(* IEC 61131-3 sources: generating_plc_code_with_llms/PLC_Code, 21 files *)

(* ---- 10.st ---- *)
FUNCTION SIGMOID : REAL
  VAR_INPUT
    X : REAL;
  END_VAR

  IF X > 20.0 THEN
  	SIGMOID := 1.0;
  ELSIF x < -85.0 THEN
  	SIGMOID := 0.0;
  ELSE
  	SIGMOID := 1.0 / (1.0 + EXP(-X));
  END_IF;
  (* from OSCAT library; www.oscat.de  *)
END_FUNCTION

(* ---- 11.st ---- *)
FUNCTION SGN : INT
  VAR_INPUT
    x : REAL;
  END_VAR

  IF X > 0.0 THEN
  	sgn := 1;
  ELSIF X < 0.0 THEN
  	sgn := -1;
  ELSE
  	sgn := 0;
  END_IF;
  (* from OSCAT library; www.oscat.de  *)
END_FUNCTION

(* ---- 12.st ---- *)
FUNCTION SINH : REAL
  VAR
    X : REAL;
  END_VAR

  IF ABS(x) < 2.0E-3 THEN
  	SINH := X;
  ELSE
  	SINH := (EXP(x) - EXP(-x)) * 0.5;
  END_IF;
  (* from OSCAT library; www.oscat.de  *)
END_FUNCTION

(* ---- 14.st ---- *)
FUNCTION FC1001 :BOOL
VAR_INPUT
	MEW: REAL;
	SP: REAL;
	HYS: REAL;
END_VAR
VAR_IN_OUT
 	OUT:BOOL;
END_VAR
VAR
 	P_HYS: REAL;
END_VAR

P_HYS:=MEW*HYS/100;
IF MEW<(SP-P_HYS/2) THEN
	OUT:=TRUE;
ELSIF
	MEW>(SP+P_HYS/2) THEN
	OUT:=FALSE;
ELSE
	OUT:=OUT;
END_IF

(* ---- 15.st ---- *)
FUNCTION FC1002 :BOOL
VAR_INPUT
	E_A, SENSOR: BOOL;
	ZEITW: TIME;
END_VAR
VAR_IN_OUT
	ZEIT:TON;
	P_HU, P_AL: BOOL;
END_VAR

IF NOT E_A THEN
	FC1002:=FALSE;
	P_HU:=FALSE;
	P_AL:=FALSE;
ELSE
	FC1002:=TRUE;
	IF P_AL THEN
		P_HU:=FALSE;
	ELSIF SENSOR THEN
		P_HU:=FALSE;
	ELSE
		P_HU:=TRUE;
	END_IF
END_IF
ZEIT(IN:=P_HU OR P_AL, PT:=ZEITW);
P_AL:=Zeit.Q;

(* ---- 18.st ---- *)
FUNCTION FC1003 : VOID
VAR_INPUT
    IN_R:REAL;
    IN_MAX, IN_MIN:REAL;
    OUT_MAX, OUT_MIN:REAL;
END_VAR
VAR_OUTPUT
    OUT_R:REAL;
    FEH:BOOL;
END_VAR
VAR_TEMP
    DIFF1, DIFF2:REAL;
END_VAR

DIFF1:= IN_MAX-IN_MIN;
DIFF2:= OUT_MAX-OUT_MIN;
FEH := (DIFF1=0) OR (DIFF2=0);
IF NOT FEH THEN
    OUT_R:= (OUT_MAX-OUT_MIN) / DIFF1 * (IN_R-IN_MIN) + OUT_MIN;
ELSE
    OUT_R:=0.0;
END_IF;
END_FUNCTION

(* ---- 2.st ---- *)
FUNCTION BINOM : INT
  VAR_INPUT
    N : INT;
    K : INT;
    i : INT;
  END_VAR

  IF 2 * K > n THEN
  	k := n - k;
  END_IF;
  IF k > n THEN
  	RETURN;
  ELSIF k = 0 OR k = n THEN
  	BINOM := 1;
  ELSIF k = 1 THEN
  	BINOM := n;
  ELSE
  	BINOM := n;
  	n := n + 1;
  	FOR i := 2 TO k DO
  		BINOM := BINOM * (n - i) / i;
  	END_FOR;
  END_IF;

END_FUNCTION

(* ---- 3.st ---- *)
FUNCTION FIB : DINT
  VAR_INPUT
    X : INT;
  END_VAR
  VAR
    t1 : DINT;
    t2 : DINT;
    x_tmp : INT;
  END_VAR

  t1 := DINT#0;
  t2 := DINT#0;
  X_tmp := X;
  IF X_tmp < 0 OR X_tmp > 46 THEN
  	FIB := DINT#-1;
  ELSIF X_tmp < 2 THEN
  	FIB := INT_TO_DINT(X_tmp);
  	RETURN;
  ELSE
  	(* the fibonacci number is the sum of the two suceeding fibonaci numbers *)
  	(* we store the numbers alternatively in t1 and t2 depending on pt *)
  	t2 := DINT#1;
  	WHILE X_tmp > 3 DO
  		X_tmp := X_tmp - 2;
  		t1 := t1 + t2;
  		t2 := t1 + t2;
  	END_WHILE;
  	IF X_tmp > 2 THEN t1 := t1 + t2; END_IF;
  	fib := t1 + t2;
  END_IF;
END_FUNCTION

(* ---- 8.st ---- *)
FUNCTION LAMBERT_W : REAL
  VAR_INPUT
    X : REAL;
  END_VAR
  VAR
    w : REAL;
    i : INT;
    we : REAL;
    w1e : REAL;
    ewx : REAL;
    last : DWORD;
  END_VAR

  IF x < -0.367879441171442 THEN
  	LAMBERT_W := -1000.0;
  	RETURN;
  (* return 0 if x = 0 *)
  ELSIF x = 0.0 THEN
  	RETURN;
  (* first an estimate is calculated *)
  ELSIF x <= 500.0 THEN
  	w := LN(x + 1.0);
  	w := 0.665 * (1.0 + 0.0195 * w) * w + 0.04;
  ELSE
  	w := LN(x - 4.0) - (1.0 - 1.0/LN(x)) * LN(LN(x));
  END_IF;
  (* use estimate to calculate exact result *)
  FOR i := 0 TO 5 DO
  	ewx := EXP(w);
  	we := w * ewx - x;
  	w1e := (w+1.0) * ewx;
  	last := REAL_TO_DWORD(w) AND DWORD#16#FFFF_FFFC;
  	w := w - (we / (w1e - (w+2.0) * we / (2.0 * w + 2.0)));
  	IF (REAL_TO_DWORD(w) AND DWORD#16#FFFF_FFFC) = last THEN EXIT; END_IF;
  END_FOR;
  LAMBERT_W := w;
  (* from OSCAT library; www.oscat.de  *)
END_FUNCTION

(* ---- 19.st ---- *)
FUNCTION_BLOCK FB1005
VAR_INPUT
    START:BOOL;
    DICKE, V_MAX, V_MIN:REAL;
END_VAR
VAR_OUTPUT
    D_MAX, D_MIN:REAL;
    P1:BOOL;
END_VAR
VAR
    FO:BOOL;
END_VAR

IF NOT START THEN
    FO:=START;
    RETURN;
END_IF;
IF START=TRUE AND FO=FALSE THEN
    D_MAX:=DICKE;
    D_MIN:=DICKE;
    P1:=FALSE;
END_IF;
FO:=START;
IF DICKE < D_MIN THEN
    D_MIN:=DICKE;
END_IF;
IF DICKE > D_MAX THEN
    D_MAX:=DICKE;
END_IF;
IF D_MIN < V_MIN OR D_MAX > V_MAX THEN
    P1:=TRUE;
END_IF;
END_FUNCTION_BLOCK

(* ---- 20.st ---- *)
FUNCTION_BLOCK INTERLOCK
    VAR_INPUT
        I1 : BOOL;
        I2 : BOOL;
        TL : TIME;
    END_VAR
    VAR_OUTPUT
        Q1 : BOOL;
        Q2 : BOOL;
    END_VAR
    VAR
        T1 : TOF;
        T2 : TOF;
    END_VAR

    T1(IN := I1, PT := TL);
    T2(IN := I2, PT := TL);

    Q1 := I1 AND NOT t2.Q;
    Q2 := I2 AND NOT t1.Q;

END_FUNCTION_BLOCK

(* ---- 21.st ---- *)
FUNCTION_BLOCK BURNER
  VAR_INPUT
    IN : BOOL;
    STAGE2 : BOOL;
    OVER_TEMP : BOOL;
    OIL_TEMP : BOOL := TRUE;
    FLAME : BOOL;
    RST : BOOL;
    RST_TIMER : BOOL;
    PRE_HEAT_TIME : TIME := t#5s;
    PRE_VENT_TIME : TIME := t#15s;
    PRE_IGNITE_TIME : TIME := t#15s;
    POST_IGNITE_TIME : TIME := t#25s;
    STAGE2_DELAY : TIME := t#10s;
    SAFETY_TIME : TIME := t#5s;
    LOCKOUT_TIME : TIME := t#10s;
    MULTIPLE_IGNITION : BOOL := TRUE;
    KW1 : REAL;
    KW2 : REAL;
  END_VAR
  VAR_OUTPUT
    MOTOR : BOOL;
    COIL1 : BOOL;
    COIL2 : BOOL;
    PRE_HEAT : BOOL;
    IGNITE : BOOL;
    FAIL : BOOL;
    KWH : REAL;
    STATUS : BYTE;
  END_VAR
  VAR_IN_OUT
    RUNTIME1 : UDINT;
    RUNTIME2 : UDINT;
    CYCLES : UDINT;
  END_VAR
  VAR
    state : INT;
    last : TIME;
    tx : TIME;
    last_change : TIME;
    timer1 : ONTIME;
    timer2 : ONTIME;
    oil_temp_last : BOOL;
    cycles2 : UDINT;
  END_VAR

  tx:= UDINT_TO_TIME(T_PLC_MS(en:=true));

  (* check rst input and overtemp *)
  IF rst OR over_temp OR state = 0 THEN
  	IF status > BYTE#0 AND tx - last_change >= lockout_time AND rst THEN
  		status := BYTE#110;
  		fail := FALSE;
  		state := 1;
  	ELSE
  		(* normaler reset *)
  		motor := FALSE;
  		coil1 := FALSE;
  		coil2 := FALSE;
  		ignite := FALSE;
  		pre_heat := FALSE;
  		IF over_temp THEN
  			status := BYTE#9;
  			fail := TRUE;
  		END_IF;
  		last_change := tx;
  		last := tx;
  		state := 1;
  	END_IF;
  END_IF;

  (* check for timer rst and rst timer if true *)
  IF rst_timer THEN
  	runtime1 := UDINT#0;
  	runtime2 := UDINT#0;
  	cycles := UDINT#0;
  	cycles2 := UDINT#0;
  END_IF;

  (* quit here if an error is present *)
  IF (status > BYTE#0 AND status < BYTE#100) OR rst THEN RETURN; END_IF;

  (* start sequence *)
  CASE state OF

  1:	(* in signal starts oil pre heating *)
  	IF in AND flame THEN
  		state := 7;
  		pre_heat := FALSE;
  		status := BYTE#2;
  		last_change := tx;
  	ELSIF in THEN
  		pre_heat := TRUE;
  		state := 2;
  		last_change := tx;
  	END_IF;

  2:	(* after pre_heating time start motor *)
  	IF (tx- last_change >= pre_heat_time AND oil_temp) OR (oil_temp AND NOT oil_temp_last) THEN
  		motor := TRUE;
  		state := 3;
  		last_change := tx;
  	(* pre_heat_time ist abgelaufen und oil_temp ist nicht aktiv *)
  	ELSIF tx - last_change >= pre_heat_time AND NOT oil_temp THEN
  		state := 7;
  		pre_heat := FALSE;
  		status := BYTE#1;
  		last_change := tx;
  	(* flame monitor cannot be active at this time *)
  	ELSIF flame THEN
  		state := 7;
  		pre_heat := FALSE;
  		status := BYTE#2;
  		last_change := tx;
  	END_IF;

  3:	(* abwarten bis zündung eingeschaltet werden kann *)
  	IF tx - last_change >= pre_vent_time - pre_ignite_time THEN
  		ignite := TRUE;
  		state := 4;
  		last_change := tx;
  	(* flame monitor cannot be active at this time *)
  	ELSIF flame THEN
  		state := 7;
  		pre_heat := FALSE;
  		motor := FALSE;
  		status := BYTE#3;
  		last_change := tx;
  	END_IF;

  4:	(* warten bis oelzufuhr geoeffnet werden darf *)
  	IF tx - last_change >= pre_ignite_time THEN
  		coil1 := TRUE;
  		state := 5;
  		last_change := tx;
  	END_IF;

  5:	(* warten auf flammwaechter und falls noetig abschalten *)
  	IF tx - last_change >= safety_time OR flame THEN
  		IF NOT flame THEN
  			(* notabschaltung da flammwaechster nicht angesprochen hat *)
  			state := 7;
  			motor := FALSE;
  			coil1 := FALSE;
  			pre_heat := FALSE;
  			ignite := FALSE;
  			status := BYTE#4;
  			last_change := tx;
  		ELSE
  			state := 6;
  			last_change := tx;
  		END_IF;
  	END_IF;

  6:	(* brenner läuft, flammueberwachung und nach ablauf der nachigniteszeit ignite abschalten *)
  	IF NOT flame AND NOT multiple_ignition THEN
  		(* notabschaltung da flammwaechster keine flamme meldet *)
  		state := 7;
  		motor := FALSE;
  		coil1 := FALSE;
  		coil2 := FALSE;
  		pre_heat := FALSE;
  		ignite := FALSE;
  		status := BYTE#5;
  		last_change := tx;
  	ELSIF NOT flame AND multiple_ignition THEN
  		ignite := TRUE;
  		state := 5;
  		coil2 := FALSE;
  		last_change := tx;
  	ELSE
  		IF tx - last_change >= post_ignite_time THEN
  			(* post_ignite_time abgelaufen, ignite abschalten *)
  			ignite := FALSE;
  		END_IF;
  		IF tx - last_change >= stage2_delay AND stage2 THEN
  			coil2 := TRUE;
  		ELSE
  			coil2 := FALSE;
  		END_IF;
  	END_IF;
  END_CASE;

  (* abschaltung wenn kein eingangssignal *)
  IF NOT in THEN
  	state := 1;
  	motor := FALSE;
  	coil1 := FALSE;
  	coil2 := FALSE;
  	ignite := FALSE;
  	pre_heat := FALSE;
  	last_change := tx;
  END_IF;

  (* runtimezähler *)
  timer1(in := flame AND in AND motor AND coil1 AND NOT coil2, SECONDS := runtime1, CYCLES := cycles);
  cycles := timer1.CYCLES;
  runtime1 := timer1.SECONDS;

  timer2(in := flame AND in AND motor AND coil1 AND coil2, SECONDS := runtime2, CYCLES := cycles2);
  cycles2 := timer2.CYCLES;
  runtime2 := timer2.SECONDS;

  KWH := UDINT_TO_REAL(runtime1) * KW1 / 3600.0 + UDINT_TO_REAL(runtime2) * KW2 / 3600.0;

  (* zeit fuer naechsten aufruf merken *)
  last := tx;

  (* set fail output IF ERROR and Status  if normal operation *)

  IF status > BYTE#0 AND status < BYTE#100 THEN
  	fail := TRUE;
  ELSE
  	fail := FALSE;
  	IF NOT in THEN
  		status := BYTE#110;
  	ELSIF flame AND in AND motor AND coil2 AND coil1 THEN
  		status := BYTE#113;
  	ELSIF flame AND in AND motor AND coil1 THEN
  		status := BYTE#112;
  	ELSE
  		status := BYTE#111;
  	END_IF;
  END_IF;

  (* From OSCAT Library, www.OSCAT.de *)
  (* T_PLC_MS, ONTIME required *)
END_FUNCTION_BLOCK

(* ---- 1.st ---- *)
VAR
	xAllOn : BOOL;
	xAllOff : BOOL;

	xAlarm1 : BOOL;
    xAlarm2 : BOOL;
END_VAR

IF xAllOn THEN
	xAllOn := FALSE;

	xAlarm1 := TRUE;
	xAlarm2 := TRUE;
END_IF

IF xAllOff THEN
	xAllOff := FALSE;

	xAlarm1 := FALSE;
    xAlarm2 := FALSE;
END_IF

(* ---- 13.st ---- *)
VAR CONSTANT
    MAXNUMBERS : UINT := 99;
END_VAR

VAR
    aNumbers : ARRAY[0..MAXNUMBERS] OF INT;
    nCnt : INT;
END_VAR

nCnt := 0;
REPEAT
    IF aNumbers[nCnt] = 10 THEN
    (*found the number 10*)
    EXIT;
    END_IF
    nCnt := nCnt + 1;
    UNTIL nCnt > MAXNUMBERS
END_REPEAT

(* ---- 16.st ---- *)
VAR
    North_green : BOOL;
    North_yellow : BOOL;
    North_red : BOOL;
    East_green : BOOL;
    East_yellow : BOOL;
    East_red : BOOL;
    T1 : TON;
END_VAR

PROGRAM traffic_light
T1.PRE := 10000;
T1.TimerEnable := 1;
T1.Reset := T1.DN

IF T1.ACC > 0 AND T1.ACC < 5000 THEN
    North_green := TRUE;
    North_yellow := FALSE;
    North_red := FALSE;
    East_green := FALSE;
    East_yellow := FALSE;
    East_red := TRUE;
END_IF

IF T1.ACC > 5000 AND T1.ACC < 5500 THEN
    North_green := FALSE;
    North_yellow := TRUE;
    North_red := FALSE;
    East_green := FALSE;
    East_yellow := FALSE;
    East_red := TRUE;
END_IF

IF T1.ACC > 5500 AND T1.ACC < 9500 THEN
    North_green := FALSE;
    North_yellow := FALSE;
    North_red := TRUE;
    East_green := TRUE;
    East_yellow := FALSE;
    East_red := FALSE;
END_IF

IF T1.ACC > 9500 AND T1.ACC < 10000 THEN
    North_green := FALSE;
    North_yellow := FALSE;
    North_red := TRUE;
    East_green := FALSE;
    East_yellow := TRUE;
    East_red := FALSE;
END_IF

END_PROGRAM

(* ---- 17.st ---- *)
VAR
    aiOutside : INT;
    aiHumidity: INT;
    sShowText : STRING[80];
END_VAR

IF aiOutside < 18 THEN
    sShowText := 'Cold';
ELSIF (aiOutside >= 18) AND (aiOutside <= 25) THEN
    IF (aiHumid >= 40) AND (aiHumid <= 75) THEN
        sShowText := 'Opt';
    ELSE
        sShowText := 'Temp. Ok';
    END_IF
ELSE
    sShowText := 'Hot';
END_IF;

(* ---- 4.st ---- *)
VAR
    aiLevel : INT;
    PercentLevel : UINT;
    doLow : BOOL;
    doOk : BOOL;
    doHigh : BOOL;
    doAlarm : BOOL;
END_VAR

(*scaling the analog input to percent*)
PercentLevel := INT_TO_UINT(aiLevel / 327);
(*reset all outputs*)
doAlarm := FALSE;
doLow := FALSE;
doOk := FALSE;
doHigh := FALSE;

CASE PercentLevel OF
    0: (*-- level alarm*)
        doAlarm := TRUE;
        doLow := TRUE;
    1..24: (*-- level is low*)
        doLow := TRUE;
    25..90:(*-- level is ok*)
        doOk := TRUE;
    ELSE (*-- level is high*)
        doHigh := TRUE;
END_CASE

(* ---- 5.st ---- *)
VAR
    Start_Loop : BOOL := FALSE;
    one_hour : TIME := T#1h;
    One_Hour_Timer : TON;
    Gate_Open : BOOL := FALSE;
    Close_Gate_Inst : BOOL := FALSE;
    Sensed_Car : BOOL := FALSE;
    Sensed_Car_Inst : BOOL := FALSE;
    Sensed_App : BOOL := FALSE;
    Mobile_Inst : BOOL := FALSE;
    Auth : STRING;
    my_defined_str : STRING := 'abcd';
END_VAR

One_Hour_Timer(IN := NOT(Start_Loop), PT := one_hour);

IF One_Hour_Timer.Q THEN
  IF Gate_Open THEN
    Close_Gate_Inst := TRUE;
    Gate_Open := FALSE;
  END_IF;
END_IF;

IF Sensed_App THEN
  IF Auth = my_defined_str THEN
    Close_Gate_Inst := Mobile_Inst XOR Gate_Open;
    Gate_Open := Mobile_Inst;
  END_IF;
END_IF;

IF Sensed_Car THEN
  IF Auth = my_defined_str THEN
    Close_Gate_Inst := Sensed_Car_Inst XOR Gate_Open;
    Gate_Open := Sensed_Car_Inst;
  END_IF;
END_IF;

Start_Loop := One_Hour_Timer.Q;

(* ---- 6.st ---- *)
VAR CONSTANT
    WAIT : UINT:= 0;
    TOP_POSITION : UINT:= 1;
    BOTTOM_POSITION : UINT:= 2;
    GETBOX : UINT:= 3;
    UNLOAD_POSITION : UINT:= 4;
    UNLOAD_BOX : UINT:= 5;
END_VAR

VAR
    (*-- digital outputs*)
    doConvTop: BOOL;
    doConvBottom: BOOL;
    doConvLift: BOOL;
    doLiftTop: BOOL;
    doLiftBottom: BOOL;
    doLiftUnload: BOOL;
    (*-- digital inputs*)
    diConvTop: BOOL;
    diConvBottom: BOOL;
    diLiftTop: BOOL;
    diLiftBottom: BOOL;
    diLiftUnload: BOOL;
    diBoxLift: BOOL;
    (*-- status variables*)
    selectLift: UINT;
    ConvTopOn: BOOL;
    ConvBottomOn: BOOL;
END_VAR

doConvTop := NOT diConvTop OR ConvTopOn;
doConvBottom := NOT diConvBottom OR ConvBottomOn;
CASE selectLift OF
    (*-- wait for request*)
    WAIT:
        IF (diConvTop = TRUE) THEN
            selectLift := TOP_POSITION;
        ELSIF (diConvBottom = TRUE) THEN
            selectLift := BOTTOM_POSITION;
        END_IF
    (*-- move lift to top position*)
    TOP_POSITION:
        doLiftTop := TRUE;
        IF (diLiftTop = TRUE) THEN
            doLiftTop := FALSE;
            ConvTopOn := TRUE;
            selectLift := GETBOX;
        END_IF
    (*-- move lift to bottom position*)
    BOTTOM_POSITION:
        doLiftBottom := TRUE;
        IF (diLiftBottom = TRUE) THEN
            doLiftBottom := FALSE;
            ConvBottomOn := TRUE;
            selectLift := GETBOX;
        END_IF
    (*-- move box to lift*)
    GETBOX:
        doConvLift := TRUE;
        IF (diBoxLift = TRUE) THEN
            doConvLift := FALSE;
            ConvTopOn := FALSE;
            ConvBottomOn := FALSE;
            selectLift := UNLOAD_POSITION;
        END_IF
    (*-- move lift to unload position*)
    UNLOAD_POSITION:
        doLiftUnload := TRUE;
        IF (diLiftUnload = TRUE) THEN
            doLiftUnload := FALSE;
            selectLift := UNLOAD_BOX;
        END_IF
    (*-- unload the box*)
    UNLOAD_BOX:
        doConvLift := TRUE;
        IF (diBoxLift = FALSE) THEN
            doConvLift := FALSE;
            selectLift := WAIT;
        END_IF
END_CASE

(* ---- 7.st ---- *)
VAR CONSTANT
    MAX_INDEX: USINT := 4;
END_VAR
VAR
    aWeights : ARRAY[0..MAX_INDEX] OF INT;
    iCnt : USINT;
    sumWeight : DINT;
    avgWeight : INT;
END_VAR

sumWeight := 0;
FOR iCnt := 0 TO MAX_INDEX DO
    sumWeight := sumWeight + aWeights[iCnt];
END_FOR
avgWeight := DINT_TO_INT (sumWeight / (MAX_INDEX + 1));

(* ---- 9.st ---- *)
VAR
    YEAR : INT
END_VAR

IF (year MOD INT#400) = INT#00 THEN
  leap_year := TRUE;
ELSIF (year MOD INT#100) = INT#00 THEN
  leap_year := FALSE;
ELSIF (year MOD INT#04) = INT#00 THEN
  leap_year := TRUE;
ELSE
  leap_year := FALSE;
END_IF;
